{attribute 'qualified_only'}
{attribute 'strict'}
TYPE DUT_ErrorState :
(
	None,
	Active,
	Inactive,
	Acknoledged
);
END_TYPE

(* stored: Version 1.1.0.1, ProductVersion 3.1.4022.6
   DUT DUT_ErrorState: Id {2803a21e-b5ef-48fc-a5fd-18043e60c6af} *)
